PROGRAM ControlGrabAuto
VAR_INPUT
	State: INT := 0;
	NewState: INT := 0;
END_VAR

VAR

	(* INTEGERS *)
	(*uiGripOffset: 		USINT := 220;			(* Offset				-->	Afstand ud til grip, når befinder sig i Home pos	-	Afstand i mm. i Y retning	*)
	uiTrunkPos: 		UINT;				(* Stamme position	-->	Afstand i mm.															*)
	iBunchPosZ: 		UINT;
	iStemAngle:		INT;

	iStemPosX: 		UINT;				(* *)
	iStemPosY: 		UINT;				(* *)
	iStemPosZ: 		UINT;
	iRoll: 			INT;
	iPitch: 			UINT;
	iYaw:			INT;
	iPickAngle: 		INT;*)

	iMoved: 			INT;					(* Hvor mange gange har cut bevæget sig efter iBundPosZ er nået *)
	iCnfgChange:		INT := 0;

	(* REALS *)

	(* Timer *)
	bJointFound: BOOL;
	bStemFound: BOOL;
	flag: BOOL;
	bStopped: BOOL;
	bAngleFlag: BOOL;
	bDeloaded: BOOL;

	uiDeleaf: UINT;
END_VAR

CASE State OF

	0:		(* init	-	Every important variables will be resat before the start of the sequence *)
		IF bStart AND uiprogNo = 5 AND State <> 2000  AND NOT bAlarmState THEN
			uiStatus := 1;

			(* Init variables *)
			uiCalibImgCount	:= 0;
			iMoved := 0;
			iImageZone := 0;
			GviX := 0;
			GviY := 0;
			GviZ := 0;
			GviA := 0;
			GviE := 0;
			GviR := 0;
			GviPick := 0;
			iPickAngle := 0;
			gResetPcCom 	:= TRUE;
			iCnfgChange := 0;
			uiDeleaf := 0;

			(* Before starting - Home *)
			GbHomeGripStem := TRUE;
			IF bHomeDone THEN
				bStart := FALSE;
				bHomeDone := FALSE;
				NewState := 10;
			END_IF
		END_IF

	10:		(* Set velocity *)
		uiSignalOutSpeedControl := UINT_TO_BYTE(uiSpeedSetting);
		FB_SET_VELOCITY.Execute := TRUE;
		uiSignalOutControl := FB_SET_VELOCITY.OutQ;
		IF FB_SET_VELOCITY.Done THEN
			FB_SET_VELOCITY.Execute := FALSE;
			NewState := 20;
		END_IF

	20:		(* Idle *)
		FB_MOVE_TO_IDLE.Execute := TRUE;
		uiSignalOutControl := FB_MOVE_TO_IDLE.OutQ;
		IF FB_MOVE_TO_IDLE.Done THEN
			FB_MOVE_TO_IDLE.Execute := FALSE;
			NewState := 30;
		END_IF

	30:		(*  Load cutter *)
		FB_LOAD_CUT.Execute := TRUE;
		IF FB_LOAD_CUT.Done THEN
			FB_LOAD_CUT.Execute := FALSE;
			NewState := 40;
		END_IF

	40: 		(* Cam 1 Take image	-	parameters recieved from Vision = height of lowest ripe tomato and Y coord for lowest point of the stem *)

		FB_CAM_ONE_CONTROL.Execute := TRUE;
		IF FB_CAM_ONE_CONTROL.Done THEN
			FB_CAM_ONE_CONTROL.Execute := FALSE;

			uiDistToGrab	:= FB_CAM_ONE_CONTROL.TrunkDist;
			iBunchPosZ 	:= FB_CAM_ONE_CONTROL.BunchHeight;
			iStemAngle	:= FB_CAM_ONE_CONTROL.StemHeading;
			iImageZone	:= FB_CAM_ONE_CONTROL.Zone;
			NewState := 50;
		END_IF

	50:		(* Joris gripper retreives stem *)
		(* Grab stem and pull in *)
		IF NOT bAck THEN
			(* HMI knap der kalder GribStem *)
			GbGripStem := TRUE;
		ELSIF bAck THEN
			gResetPcCom := TRUE;
			NewState := 55;
		END_IF

	55:
		IF uiToolState = 0 THEN
			NewState := 100;
		END_IF

	(* ---------------------------- Grab the stem ---------------------------- *)

	100:		(* Robot Pick move to Image Pos *)
		FB_PICK_TRUNK_IMAGE.Execute := TRUE;
		uiSignalOutControl := FB_PICK_TRUNK_IMAGE.OutQ;
		IF FB_PICK_TRUNK_IMAGE.Done THEN
			FB_PICK_TRUNK_IMAGE.Execute := FALSE;
			gResetPcCom := TRUE;
			NewState := 110;
		END_IF

	110:		(* Send Robot Pick Position *)
		getPickCoords := TRUE;
		IF bPosSentToPcCom AND FB_GET_PICK_COORD.Execute = FALSE THEN
			bPosSentToPcCom := FALSE;
			bGetCoordDone := FALSE;
			NewState := 120;
		END_IF

	120:		(* Cam 2 take image *)
		(* Take bottom Image *)
		IF stDataToVision.CoordXR2G <> 0 AND stDataToVision.CoordYR2G <> 0 AND stDataToVision.CoordZR2G <> 0 THEN
			FB_CAM_TWO_CONTROL.Execute := TRUE;
			IF FB_CAM_TWO_CONTROL.Done THEN
				FB_CAM_TWO_CONTROL.Execute := FALSE;
				IF FB_CAM_TWO_CONTROL.X > 420 OR FB_CAM_TWO_CONTROL.X < 125 OR FB_CAM_TWO_CONTROL.Y > 400 OR FB_CAM_TWO_CONTROL.Y < 125 THEN
					NewState := 1000;
				ELSE
					GviX := FB_CAM_TWO_CONTROL.X;
					GviY := FB_CAM_TWO_CONTROL.Y;
					GviZ := FB_CAM_TWO_CONTROL.Z;
					GviA := FB_CAM_TWO_CONTROL.RotZ0;
					GviE := FB_CAM_TWO_CONTROL.RotY;
					GviR := FB_CAM_TWO_CONTROL.RotZ1;
					gResetPcCom := TRUE;
					NewState := 130;
				END_IF
			END_IF
		END_IF

	130:		(* Send Pos to Robot *)

		(* GsendCoord			-->	Starter SendCoordinates sekvensen							-	Sender koordinater til robotterne 		*)
		(* uiSignalOutShared.06	-->	Bekræftelse på at koordinaterne er sendt til udgangene i box 10	-	Acknowledge fra SendCoordinates	*)
		GsendCoord := TRUE;
		IF uiSignalOutShared.06 THEN
			(* Send_pos	-->	Kommando der fortæller robot cut at nogle nye positioner er sendt *)
			uiSignalOutControl := Send_pos;
		END_IF
		IF uiSignalInAck = Send_pos THEN
			uiSignalOutControl := 0;
			uiCalibImgCount := uiCalibImgCount + 1;
			NewState := 135;
		END_IF

	135:
		IF uiSignalInAck = 0 THEN
			NewState := 140;
		END_IF

	140:		(* Move Pick to next image pos *)
		FB_PICK_TRUNK_IMAGE.Execute := TRUE;
		uiSignalOutControl := FB_PICK_TRUNK_IMAGE.OutQ;
		IF FB_PICK_TRUNK_IMAGE.Done THEN
			FB_PICK_TRUNK_IMAGE.Execute := FALSE;
			NewState := 150;
		END_IF

	150:		(* Send Pick pos to PcCom for next image *)
		getPickCoords := TRUE;
		IF bPosSentToPcCom AND FB_GET_PICK_COORD.Execute = FALSE THEN
			bPosSentToPcCom := FALSE;
			bGetCoordDone := FALSE;
			NewState := 160;
		END_IF

	160:		(* Move Cut to Stem *)
		FB_CUT_TO_STEM.Execute := TRUE;
		uiSignalOutControl := FB_CUT_TO_STEM.OutQ;
		IF FB_CUT_TO_STEM.Done THEN
			FB_CUT_TO_STEM.Execute := FALSE;
			IF FB_CAM_TWO_CONTROL.Z >= iBunchPosZ THEN
				NewState := 300;
			ELSE
				NewState := 200;
			END_IF
		END_IF

		(* ------------------------------------------ Move on stem ------------------------------------------ *)

	200:		(* Cam 2: Take new Image *)
		IF stDataToVision.CoordXR2G <> 0 AND stDataToVision.CoordYR2G <> 0 AND stDataToVision.CoordZR2G <> 0 THEN
			FB_CAM_TWO_CONTROL.Execute := TRUE;
			IF FB_CAM_TWO_CONTROL.Done THEN
				FB_CAM_TWO_CONTROL.Execute := FALSE;
				IF FB_CAM_TWO_CONTROL.StemFound = 1 THEN
					IF FB_CAM_TWO_CONTROL.X > 500 OR FB_CAM_TWO_CONTROL.X < 125 OR FB_CAM_TWO_CONTROL.Y > 425 OR FB_CAM_TWO_CONTROL.Y < 125 THEN
						NewState := 1000;
					ELSE
						GviX := FB_CAM_TWO_CONTROL.X;
						GviY := FB_CAM_TWO_CONTROL.Y;
						GviZ := FB_CAM_TWO_CONTROL.Z;
						GviA := 0;
						GviE := 0;
						GviR := 40;
						IF FB_CAM_TWO_CONTROL.JointFound = 1 THEN
							GviPick := FB_CAM_TWO_CONTROL.PickAngle;
							iImageZone := FB_CAM_TWO_CONTROL.Zone;
							gResetPcCom := TRUE;
							NewState := 310;
						ELSE
							gResetPcCom := TRUE;
							NewState := 210;
						END_IF
					END_IF
				ELSE
					gResetPcCom := TRUE;
					NewState := 345;
				END_IF
			END_IF
		END_IF

	210:		(* Send pos to Robots *)
		(* GsendCoord			-->	Starter SendCoordinates sekvensen							-	Sender koordinater til robotterne 		*)
		(* uiSignalOutShared.06	-->	Bekræftelse på at koordinaterne er sendt til udgangene i box 10	-	Acknowledge fra SendCoordinates	*)
		GsendCoord := TRUE;
		IF uiSignalOutShared.06 THEN
			(* Send_pos	-->	Kommando der fortæller robot cut at nogle nye positioner er sendt *)
			uiSignalOutControl := Send_pos;
		END_IF
		IF uiSignalInAck = Send_pos THEN
			uiSignalOutControl := 0;
			uiCalibImgCount := uiCalibImgCount + 1;
			NewState := 215;
		END_IF

	215:
		IF uiSignalInAck = 0 THEN
			NewState := 220;
		END_IF

	220:		(* Robot Pick to image pos *)
		FB_PICK_TRUNK_IMAGE.Execute := TRUE;
		uiSignalOutControl := FB_PICK_TRUNK_IMAGE.OutQ;
		IF FB_PICK_TRUNK_IMAGE.Done THEN
			FB_PICK_TRUNK_IMAGE.Execute := FALSE;
			NewState := 230;
		END_IF

	230: 		(* Send Pick coordinate *)
		(* Send Pick pos to PcCom for next image *)
		getPickCoords := TRUE;
		IF bPosSentToPcCom AND FB_GET_PICK_COORD.Execute = FALSE THEN
			bPosSentToPcCom := FALSE;
			NewState := 240;
		END_IF

	240:		(* Move cut on stem *)
		FB_CUT_ON_STEM.Execute := TRUE;
		uiSignalOutControl := FB_CUT_ON_STEM.OutQ;
		(* MOVE_TO_STEM bliver sendt tilbage som bekræftelse *)
		IF FB_CUT_ON_STEM.Done THEN
			FB_CUT_ON_STEM.Execute := FALSE;
			IF iStemPosZ >= iBunchPosZ THEN
				iMoved := 0;
				NewState := 300;
			ELSE
				NewState := 200;
			END_IF
		END_IF

	(* ------------------------------------------ Find Joint ------------------------------------------ *)

	300:		(* Take a picture *)
		IF stDataToVision.CoordXR2G <> 0 AND stDataToVision.CoordYR2G <> 0 AND stDataToVision.CoordZR2G <> 0 THEN
			FB_CAM_TWO_CONTROL.Execute := TRUE;
			IF FB_CAM_TWO_CONTROL.Done THEN
				FB_CAM_TWO_CONTROL.Execute := FALSE;
				IF FB_CAM_TWO_CONTROL.StemFound = 1 THEN
					IF FB_CAM_TWO_CONTROL.X > 500 OR FB_CAM_TWO_CONTROL.X < 125 OR FB_CAM_TWO_CONTROL.Y > 425 OR FB_CAM_TWO_CONTROL.Y < 125 THEN
						NewState := 1000;
					ELSE
						GviPick := FB_CAM_TWO_CONTROL.PickAngle;
						IF FB_CAM_TWO_CONTROL.Zone <> 0 THEN
							iImageZone := FB_CAM_TWO_CONTROL.Zone;
						END_IF
						IF FB_CAM_TWO_CONTROL.JointFound = 1 THEN
							GviPick := FB_CAM_TWO_CONTROL.PickAngle;
						ELSE
							GviX := FB_CAM_TWO_CONTROL.X;
							GviY := FB_CAM_TWO_CONTROL.Y;
							GviZ := FB_CAM_TWO_CONTROL.Z;
							GviA := 0;
							GviE := 0;
							GviR := 40;
						END_IF
						gResetPcCom := TRUE;
						NewState := 310;
					END_IF
				ELSE
					gResetPcCom := TRUE;
					NewState := 345;
				END_IF
			END_IF
		END_IF

	310:		(* Send pos *)
		(* GsendCoord			-->	Starter SendCoordinates sekvensen							-	Sender koordinater til robotterne 		*)
		(* uiSignalOutShared.06	-->	Bekræftelse på at koordinaterne er sendt til udgangene i box 10	-	Acknowledge fra SendCoordinates	*)
		GsendCoord := TRUE;
		IF uiSignalOutShared.06 THEN
			(* Send_pos	-->	Kommando der fortæller robot cut at nogle nye positioner er sendt *)
			uiSignalOutControl := Send_pos;
		END_IF
		IF uiSignalInAck = Send_pos THEN
			uiSignalOutControl := 0;
			uiCalibImgCount := uiCalibImgCount + 1;
			bAngleFlag := FALSE;
			NewState := 315;
		END_IF

	315:
		IF uiSignalInAck = 0 THEN
			IF FB_CAM_TWO_CONTROL.JointFound = 1 THEN
				NewState := 345;
			ELSE
				NewState := 320;
			END_IF
		END_IF

	320:		(* Pick image pos *)
		(* Robot Pick to image pos *)
		FB_PICK_TRUNK_IMAGE.Execute := TRUE;
		uiSignalOutControl := FB_PICK_TRUNK_IMAGE.OutQ;
		IF FB_PICK_TRUNK_IMAGE.Done THEN
			FB_PICK_TRUNK_IMAGE.Execute := FALSE;
			NewState := 330;
		END_IF

	330: 		(* Send Pick coordinate *)
		(* Send Pick pos to PcCom for next image *)
		getPickCoords := TRUE;
		IF bPosSentToPcCom AND FB_GET_PICK_COORD.Execute = FALSE THEN
			bPosSentToPcCom := FALSE;
			NewState := 340;
		END_IF

	340:		(* Move on Stem *)
		FB_CUT_ON_STEM.Execute := TRUE;
		uiSignalOutControl := FB_CUT_ON_STEM.OutQ;
		(* MOVE_TO_STEM bliver sendt tilbage som bekræftelse *)
		IF FB_CUT_ON_STEM.Done THEN
			FB_CUT_ON_STEM.Execute := FALSE;
			iCnfgChange := 0;
			iMoved := iMoved +1;
			NewState := 345;
		END_IF

	345:
		IF uiSignalInAck = 0 THEN
			IF stDataFromVision.gJointFound = 1  THEN
				(* Grabbing sequence *)
				gResetPcCom := TRUE;
				NewState := 400;
			ELSIF stDataFromVision.gStemFound = 1 AND stDataFromVision.gJointFound = 0 AND iMoved < 2 THEN
				(* Move further Along stem *)
				NewState := 300;
			ELSIF stDataFromVision.gStemFound = 0 OR iMoved >= 2 THEN
				(* Change configuration *)
				iCnfgChange := iCnfgChange + 1;
				IF uiCalibImgCount >= 50 AND uiCalibImgCount <= 200 THEN
					NewState := 350;
				ELSIF uiCalibImgCount = 250 THEN
					NewState := 450;
				END_IF
				gResetPcCom := TRUE;
				NewState := 350;
			ELSIF stDataFromVision.gJointFound = 255 THEN 	(* If timeout *)
				NewState := 1000;
			END_IF
		END_IF

	(* ------------------------------------------ Change configuration ------------------------------------------ *)
	350:
		IF iCnfgChange <= 5 THEN
			uiCalibImgCount := INT_TO_BYTE(iCnfgChange * 50);
		ELSE
			NewState := 600;
		END_IF
		(* Robot Pick to image pos *)
		FB_PICK_TRUNK_IMAGE.Execute := TRUE;
		uiSignalOutControl := FB_PICK_TRUNK_IMAGE.OutQ;
		IF FB_PICK_TRUNK_IMAGE.Done THEN
			FB_PICK_TRUNK_IMAGE.Execute := FALSE;
			NewState := 360;
		END_IF

	360:		(* Send Pick coordinate *)
		(* Send Pick pos to PcCom for next image *)
		getPickCoords := TRUE;
		IF bPosSentToPcCom THEN
			bPosSentToPcCom := FALSE;
			NewState := 300;
		END_IF


	(* ------------------------------------------ Grab tomatoes ------------------------------------------ *)
	400:		(* Robot Pick grab *)
		FB_PICK_GRAB.Execute := TRUE;
		uiSignalOutControl := FB_PICK_GRAB.OutQ;
		IF FB_PICK_GRAB.Done THEN
			FB_PICK_GRAB.Execute := FALSE;
			NewState := 420;
		END_IF

	420:		(* Cut *)
		FB_RELEASE_CUT.Execute := TRUE;
		IF FB_RELEASE_CUT.Done THEN
			FB_RELEASE_CUT.Execute := FALSE;
			NewState := 425;
		END_IF

	425:		(* Load Cut *)
		FB_LOAD_CUT.Execute := TRUE;
		IF FB_LOAD_CUT.Done THEN
			FB_LOAD_CUT.Execute := FALSE;
			NewState := 430;
		END_IF

	430:		(* Move from pick *)
		FB_PICK_MOVE_FROM_PICK.Execute := TRUE;
		uiSignalOutControl := FB_PICK_MOVE_FROM_PICK.OutQ;
		IF FB_PICK_MOVE_FROM_PICK.Done THEN
			FB_PICK_MOVE_FROM_PICK.Execute := FALSE;
			iMoved := 1;
			NewState := 500;
		END_IF

	(* --------------------------------- DELEAFING ------------------------------------ *)
	500:		(* Image of LEAFS *)
		uiCalibImgCount := INT_TO_BYTE(iMoved * 50);
		FB_PICK_DELEAF_PROGRAM.Execute := TRUE;
		uiSignalOutControl := FB_PICK_DELEAF_PROGRAM.OutQ;
		IF FB_PICK_DELEAF_PROGRAM.Done THEN
			iMoved := iMoved + 1;
			FB_PICK_DELEAF_PROGRAM.Execute := FALSE;
			NewState := 520;
		END_IF

	520:		(* Send Pick coordinate *)
		getPickCoords := TRUE;
		IF bPosSentToPcCom AND FB_GET_PICK_COORD.Execute = FALSE THEN
			bPosSentToPcCom := FALSE;
			NewState := 530;
		END_IF

	530:
		IF stDataToVision.CoordXR2G <> 0 AND stDataToVision.CoordYR2G <> 0 AND stDataToVision.CoordZR2G <> 0 THEN
			FB_CAM_TWO_CONTROL.Execute := TRUE;
			IF FB_CAM_TWO_CONTROL.Done THEN
				FB_CAM_TWO_CONTROL.Execute := FALSE;

				IF FB_CAM_TWO_CONTROL.StemFound = 1 THEN
					IF FB_CAM_TWO_CONTROL.X > 500 OR FB_CAM_TWO_CONTROL.X < 125 OR FB_CAM_TWO_CONTROL.Y > 425 OR FB_CAM_TWO_CONTROL.Y < 125 THEN
						NewState := 1000;
					ELSE
						IF FB_CAM_TWO_CONTROL.JointFound = 1 THEN
							GviX := FB_CAM_TWO_CONTROL.X;
							GviY := FB_CAM_TWO_CONTROL.Y;
							GviZ := FB_CAM_TWO_CONTROL.Z;
							GviA := 0;
							GviE := 0;
							GviR := 40;
							GviPick := FB_CAM_TWO_CONTROL.PickAngle;
							iImageZone := FB_CAM_TWO_CONTROL.Zone;
							gResetPcCom := TRUE;
							NewState := 540;
						ELSE
							gResetPcCom := TRUE;
							NewState := 500;
						END_IF
					END_IF
				ELSIF iMoved > 3 THEN
					gResetPcCom := TRUE;
					NewState := 540;

				ELSE
					gResetPcCom := TRUE;
					NewState := 500;
				END_IF
			END_IF
		END_IF

	540:		(* Cut move on stem *)
		FB_PICK_PLACE.Execute := TRUE;
		uiSignalOutControl := FB_PICK_PLACE.OutQ;
		IF FB_PICK_PLACE.Done THEN
			FB_PICK_PLACE.Execute := FALSE;
			stDataToVision.ResultRead := 0;
			gResetPcCom := TRUE;
			IF FB_CAM_TWO_CONTROL.JointFound = 0 THEN
				NewState := 600;
			ELSE
				NewState := 550;
			END_IF
		END_IF

	550:		(* Send pos *)

		(* GsendCoord			-->	Starter SendCoordinates sekvensen							-	Sender koordinater til robotterne 		*)
		(* uiSignalOutShared.06	-->	Bekræftelse på at koordinaterne er sendt til udgangene i box 10	-	Acknowledge fra SendCoordinates	*)
		GsendCoord := TRUE;
		IF uiSignalOutShared.06 THEN
			(* Send_pos	-->	Kommando der fortæller robot cut at nogle nye positioner er sendt *)
			uiSignalOutControl := Send_pos;
		END_IF
		IF uiSignalInAck = Send_pos THEN
			uiSignalOutControl := 0;
			uiCalibImgCount := uiCalibImgCount + 1;
			NewState := 560;
		END_IF
	560:
		FB_CUT_ON_STEM.Execute := TRUE;
		uiSignalOutControl := FB_CUT_ON_STEM.OutQ;
		IF FB_CUT_ON_STEM.Done THEN
			FB_CUT_ON_STEM.Execute := FALSE;
			NewState := 570;
		END_IF

	570:		(* CUT *)
		FB_RELEASE_CUT.Execute := TRUE;
		IF FB_RELEASE_CUT.Done THEN
			FB_RELEASE_CUT.Execute := FALSE;
			NewState := 580;
		END_IF

	580:		(* Load Cut *)
		FB_LOAD_CUT.Execute := TRUE;
		IF FB_LOAD_CUT.Done THEN
			FB_LOAD_CUT.Execute := FALSE;
			NewState := 585;
		END_IF

	585:
		IF uiDeleaf < 0 THEN
			uiDeleaf := uiDeleaf + 1;
			NewState := 500;
		ELSE
			uiDeleaf := 0;
			NewState := 600;
		END_IF

	600:		(*Open Cut*)
		FB_OPEN_CUT.Execute := TRUE;
		IF FB_OPEN_CUT.Done THEN
			FB_OPEN_CUT.Execute := FALSE;
			NewState := 610;
		END_IF

	610:		(*Move cut away from stem*)
		FB_CUT_FROM_STEM.Execute := TRUE;
		uiSignalOutControl := FB_CUT_FROM_STEM.OutQ;
		IF FB_CUT_FROM_STEM.Done THEN
			FB_CUT_FROM_STEM.Execute := FALSE;
			NewState := 620;
		END_IF


	620:		(* GbReleaseStem *)
		(* Grab stem and pull in *)
		IF NOT bAck THEN
			(* HMI knap der kalder GribStem *)
			GbReleaseStem := TRUE;
		ELSIF bAck THEN
			NewState := 630;
		END_IF

	630:		(* Move to idle *)
		FB_MOVE_TO_IDLE.Execute := TRUE;
		uiSignalOutControl := FB_MOVE_TO_IDLE.OutQ;
		IF FB_MOVE_TO_IDLE.Done THEN
			FB_MOVE_TO_IDLE.Execute := FALSE;
			uiStatus := 0;
			NewState := 640;
		END_IF

	640:		(* Deload *)

		FB_DELOAD_CUT.Execute := TRUE;
		IF FB_DELOAD_CUT.Done THEN
			FB_DELOAD_CUT.Execute := FALSE;
			NewState := 0;
		END_IF



	1000:	(* Reset *)
		uiSignalOutControl  := 0;		(* Stop sequences on ROBOTS *)
		FB_CAM_ONE_CONTROL.	Execute := FALSE;
		FB_CAM_TWO_CONTROL.	Execute := FALSE;
		(* Reset timers *)
		stDataToVision.ResultRead := 1;
		gResetPcCom := TRUE;
		bDeloaded := FALSE;
		iCnfgChange := 1;
		uiCalibImgCount := 0;
		uiDeleaf := 0;
		NewState := 0;

	2000:
		bStopped := TRUE;

END_CASE

IF State <> 2000 THEN
	bStopped := FALSE;
END_IF

END_PROGRAM

(* stored: Version 1.1.0.1, ProductVersion 3.1.4022.18
   POU ControlGrabAuto: Id {432238d5-955a-4eb7-88d3-39d7468e2a05}, SpecialFunc None *)
